// TIA Portal V17 export
// export: Created 2024-08-26T21:10:48.5721235Z, ExportSetting WithDefaults, DisplayName Totally Integrated Automation Portal, DisplayVersion V17 Update 7, DisplayName TIA Portal Openness, DisplayVersion V17 Update 7, DisplayName TIA Portal Version Control Interface, DisplayVersion V17, DisplayName SINAMICS Startdrive Advanced, DisplayVersion V17 SP2, DisplayName SINAMICS Startdrive G110M, G120, G120C, G120D, G120P, G115D, DisplayVersion V17 SP2, DisplayName SINAMICS Startdrive G130, G150, S120, S150, SINAMICS MV, S210, DisplayVersion V17 SP2, DisplayName STEP 7 Professional, DisplayVersion V17 Update 7, DisplayName STEP 7 Safety, DisplayVersion V17 Update 6, DisplayName WinCC Advanced / Unified PC, DisplayVersion V17 Update 7
DATA_BLOCK "DB_EKS"   // DB305
{ S7_Optimized_Access := 'FALSE' }
VERSION : 0.1
// stored: AutoNumber false, DBAccessibleFromOPCUA true, DBAccessibleFromWebserver true, IsOnlyStoredInLoadMemory false, IsWriteProtectedInAS false
   VAR RETAIN
      STAT : Struct
         OPERATOR : Bool := TRUE;
         GAP_LEADER : Bool := TRUE;
         MAINTENANCE : Bool := TRUE;
         ADMINISTRATOR : Bool := TRUE;
         _4 : Bool := FALSE;
         _5 : Bool := FALSE;
         _6 : Bool := FALSE;
         _7 : Bool := FALSE;
         ADD_MODE_ENABLED : Bool := TRUE;
         ADD_MODE : Bool := FALSE;
         RESET : Bool := FALSE;
         NB_MAX_ACHIEVED : Bool := FALSE;
         FP_STORE_KEY_IN : Bool := FALSE;
         _15 : Bool := FALSE;
         _16 : Bool := FALSE;
         _17 : Bool := FALSE;
      END_STRUCT;
      HMI : Struct
         OPERATOR_KEY : Bool := FALSE;
         ADD_MODE : Bool := FALSE;
         END_ADD_MODE : Bool := FALSE;
         WRITE_NEW_KEY_LEVEL : Bool := FALSE;
         WRITE_NEW_KEY_ID : Bool := FALSE;
         UPDATE_NB_ADMIN : Bool := FALSE;
         _6 : Bool := FALSE;
         _7 : Bool := FALSE;
         _10 : Bool := FALSE;
         _11 : Bool := FALSE;
         _12 : Bool := FALSE;
         _13 : Bool := FALSE;
         _14 : Bool := FALSE;
         _15 : Bool := FALSE;
         _16 : Bool := FALSE;
         _17 : Bool := FALSE;
      END_STRUCT;
      TIM : Struct
         RESET_SET : Int := 9999;
         RESET_STAT : Int := 2960;
      END_STRUCT;
      PAGE_INDEX : Int := 1;   // Index of the page of HMI
      SAVE_LINE : Int := 0;   // Line to save key
      REMOVE_LINE : Int := 0;   // Line to remove key
      ACTUAL_LEVEL : Int := 5;   // Actual level of key
      NB_ADMIN : Int := 27414;   // Number of admin counted
      T_CYCLE : Int := 0;   // Index for function Cycle (look for key)
      NB_MAX_ADMIN : Int := 5;   // Number of administrator max
      Number_page_saved : Word := 16#0001;
      _res : Array[22..47] of Byte;   // Reserve
      INSERTED_KEY { S7_SetPoint := 'True'} : "udt_EKS_KEY";   // Information of Key Inserted
      HMI_PAGE { S7_SetPoint := 'True'} : Array[1..10] of "udt_EKS_KEY";   // Information displayed on HMI
      _res_1 : Array[270..299] of Byte;   // Reserve
      KEYS { S7_SetPoint := 'True'} : Array[1..130] of "udt_EKS_KEY";
      DELETE_KEY : "udt_EKS_KEY";
   END_VAR
BEGIN
   _res[22..47] := 16#00;
   INSERTED_KEY.ID1 := 16#383E_0010;
   INSERTED_KEY.ID2 := 16#3200_0000;
   INSERTED_KEY.EMPLOYEE_ID := 16#0000_0000;
   INSERTED_KEY.LEVEL := 5;
   INSERTED_KEY.COMMENTS := WSTRING#'LIMON';
   INSERTED_KEY._res_1 := 0;
   HMI_PAGE[1].ID1 := 16#2B2F_0010;
   HMI_PAGE[2].ID1 := 16#28A5_0010;
   HMI_PAGE[3].ID1 := 16#0000_0000;
   HMI_PAGE[4].ID1 := 16#71A6_0010;
   HMI_PAGE[5].ID1 := 16#8037_0010;
   HMI_PAGE[6].ID1 := 16#383E_0010;
   HMI_PAGE[7].ID1 := 16#5A1E_0010;
   HMI_PAGE[8].ID1 := 16#D65A_0010;
   HMI_PAGE[9..10].ID1 := 16#0000_0000;
   HMI_PAGE[1..2].ID2 := 16#3200_0000;
   HMI_PAGE[3].ID2 := 16#0000_0000;
   HMI_PAGE[4..8].ID2 := 16#3200_0000;
   HMI_PAGE[9..10].ID2 := 16#0000_0000;
   HMI_PAGE[1..7].EMPLOYEE_ID := 16#0000_0000;
   HMI_PAGE[8].EMPLOYEE_ID := 16#0000_0001;
   HMI_PAGE[9..10].EMPLOYEE_ID := 16#0000_0000;
   HMI_PAGE[1].LEVEL := 5;
   HMI_PAGE[2].LEVEL := 3;
   HMI_PAGE[3].LEVEL := 0;
   HMI_PAGE[4].LEVEL := 2;
   HMI_PAGE[5].LEVEL := 3;
   HMI_PAGE[6].LEVEL := 5;
   HMI_PAGE[7].LEVEL := 3;
   HMI_PAGE[8].LEVEL := 2;
   HMI_PAGE[9..10].LEVEL := 0;
   HMI_PAGE[1].COMMENTS := WSTRING#'CLAUDIO';
   HMI_PAGE[2].COMMENTS := WSTRING#'CLAUDIO-M';
   HMI_PAGE[3].COMMENTS := WSTRING#'';
   HMI_PAGE[4].COMMENTS := WSTRING#'GAP-1';
   HMI_PAGE[5].COMMENTS := WSTRING#'MANT-1';
   HMI_PAGE[6].COMMENTS := WSTRING#'LIMON';
   HMI_PAGE[7].COMMENTS := WSTRING#'MANT';
   HMI_PAGE[8].COMMENTS := WSTRING#'GAP';
   HMI_PAGE[9..10].COMMENTS := WSTRING#'';
   HMI_PAGE[1..10]._res_1 := 0;
   _res_1[270..299] := 16#00;
   KEYS[1].ID1 := 16#2B2F_0010;
   KEYS[2].ID1 := 16#28A5_0010;
   KEYS[3].ID1 := 16#0000_0000;
   KEYS[4].ID1 := 16#71A6_0010;
   KEYS[5].ID1 := 16#8037_0010;
   KEYS[6].ID1 := 16#383E_0010;
   KEYS[7].ID1 := 16#5A1E_0010;
   KEYS[8].ID1 := 16#D65A_0010;
   KEYS[9..109].ID1 := 16#0000_0000;
   KEYS[110].ID1 := 16#DB52_0010;
   KEYS[111..130].ID1 := 16#0000_0000;
   KEYS[1..2].ID2 := 16#3200_0000;
   KEYS[3].ID2 := 16#0000_0000;
   KEYS[4..8].ID2 := 16#3200_0000;
   KEYS[9..109].ID2 := 16#0000_0000;
   KEYS[110].ID2 := 16#3200_0000;
   KEYS[111..130].ID2 := 16#0000_0000;
   KEYS[1..7].EMPLOYEE_ID := 16#0000_0000;
   KEYS[8].EMPLOYEE_ID := 16#0000_0001;
   KEYS[9..130].EMPLOYEE_ID := 16#0000_0000;
   KEYS[1].LEVEL := 5;
   KEYS[2].LEVEL := 3;
   KEYS[3].LEVEL := 0;
   KEYS[4].LEVEL := 2;
   KEYS[5].LEVEL := 3;
   KEYS[6].LEVEL := 5;
   KEYS[7].LEVEL := 3;
   KEYS[8].LEVEL := 2;
   KEYS[9..109].LEVEL := 0;
   KEYS[110].LEVEL := 5;
   KEYS[111..130].LEVEL := 0;
   KEYS[1].COMMENTS := WSTRING#'CLAUDIO';
   KEYS[2].COMMENTS := WSTRING#'CLAUDIO-M';
   KEYS[3].COMMENTS := WSTRING#'';
   KEYS[4].COMMENTS := WSTRING#'GAP-1';
   KEYS[5].COMMENTS := WSTRING#'MANT-1';
   KEYS[6].COMMENTS := WSTRING#'LIMON';
   KEYS[7].COMMENTS := WSTRING#'MANT';
   KEYS[8].COMMENTS := WSTRING#'GAP';
   KEYS[9..109].COMMENTS := WSTRING#'';
   KEYS[110].COMMENTS := WSTRING#'Robins';
   KEYS[111..130].COMMENTS := WSTRING#'';
   KEYS[1..130]._res_1 := 0;
   DELETE_KEY.ID1 := 16#0000_0000;
   DELETE_KEY.ID2 := 16#0000_0000;
   DELETE_KEY.EMPLOYEE_ID := 16#0000_0000;
   DELETE_KEY.LEVEL := 0;
   DELETE_KEY.COMMENTS := WSTRING#'';
   DELETE_KEY._res_1 := 0;
END_DATA_BLOCK
